SYSTEM TEST_ARRAY_IO (* Test ARRAY_IN,ARRAY_OUT *)
  (* Standard: 61499-2 *)
  (* Version 0.0, 2000-05-27, JHC, Rockwell Automation *)
  DEVICE ARRAY_IO : FRAME_DEVICE(BOUNDS := [100,100,200,100], GRID := [1,1])
    RESOURCE RES1 : PANEL_RESOURCE
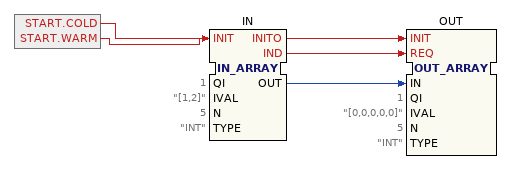
      FBS
        IN : IN_ARRAY(QI := 1, IVAL := "[1,2]", N := 5, TYPE := "INT");
        OUT : OUT_ARRAY(QI := 1, IVAL := "[0,0,0,0,0]", N := 5, TYPE := "INT");
      END_FBS
      EVENT_CONNECTIONS
        START.COLD TO IN.INIT;
        START.WARM TO IN.INIT;
        IN.INITO TO OUT.INIT;
        IN.IND TO OUT.REQ;
      END_CONNECTIONS
      DATA_CONNECTIONS
        IN.OUT TO OUT.IN;
      END_CONNECTIONS
    END_RESOURCE
  END_DEVICE
END_SYSTEM
